FUNCTION_BLOCK TcaTrolley EXTENDS TcoCore.TcoComponent

VAR CONSTANT
	MAX_CARRIERPLACES : INT := 63;
END_VAR


VAR PERSISTENT
	_data : TcaTrolleyData;
END_VAR

PROPERTY Data : REFERENCE TO TcaTrolleyData
GET
Data REF= _data;
END_GET
SET
_data := Data;
END_SET
END_PROPERTY

{warning 'Methodenimplementierung hinzufügen'}
METHOD Restore : TcoCore.ITcoRestorable
END_METHOD

{warning 'Methodenimplementierung hinzufügen'}
(*~
	<docu>
		<summary>
		    Custom service (manual, maintenance) logic.
			This method must be implemented in derived class.
		</summary>			
	</docu>	
~*)
METHOD PROTECTED ServiceMode
END_METHOD

END_FUNCTION_BLOCK

(* stored: Version 1.1.0.1
   POU TcaTrolley: Id {f529d72a-4dd4-4b6b-8f26-524d47f7e88a}, SpecialFunc None
   Property Data: Id {83c5109e-419f-447d-8e5c-89b732984431}
   Get Get: Id {ea7d11fb-c7ac-48f9-a6e1-fbf3a4992164}
   Set Set: Id {813e5464-04f3-4883-8a7d-df90c0cd049a}
   Method Restore: Id {d48b6476-49af-43a2-8ee6-0d18ee96d012}
   Method ServiceMode: Id {0366d0b8-be6d-4911-9590-379d02ca1371} *)
